TYPE ONE_BIT :
STRUCT
	e1 : BIT;
END_STRUCT
END_TYPE

(* stored: Version 1.1.0.1, ProductVersion 3.1.4024.11
   DUT ONE_BIT: Id {4f3f6d8d-7fe3-4b16-bafd-fec1946c7f65} *)
